FUNCTION_BLOCK Valve
VAR_INPUT
	//configaracionParammetr : configaracionParammetrs;
END_VAR
VAR		
	
	enaNegDir : BOOL := FALSE;
	enaPosDir : BOOL := FALSE;
	command : REAL; // Příkaz -1000 .. 0 .. 1000 [procenta * 10]

	errorDir : BOOL;
	
	currentCommand : REAL := 0;
	prolaz : STRING;
	previousenaNegDir : BOOL; 
	previousenaPosDir : BOOL;
	currentError : BOOL := FALSE; // test error
	
	//command : INT; 
	status : REFERENCE TO Staus REF=generalVariable.staus;
	konfiguraParametry : REFERENCE TO configaracionParammetrs  REF=generalVariable.conParammetr;
	speedRamp : REAL;
	
END_VAR
VAR_OUTPUT
	OutPosDir : REAL := 0 ;	// Výstup v daném směru [mA]
	OutNegDir : REAL := 0 ;	// Výstup v daném směru [mA]
END_VAR

//currentDir := currentDirB(enaNegDir,enaPosDir);
signalStandstill();
prolaz := 'fb';
IF (currentcommand <> command) THEN
		//nTime := elapsTime(direction := currentDir);
		prolaz := 'različiti';
		currentcommand := rampValve ();
	ELSE	
		Accel_Decel(FALSE, FALSE);
		status.bDone := TRUE;
END_IF;

METHOD PRIVATE Accel_Decel
VAR_INPUT
	a : BOOL;
	b : BOOL;
END_VAR
status.Accel := a;
status.Decel := b;
END_METHOD

METHOD addCommand
VAR_INPUT
	comm : real;
END_VAR
command := comm;	
currentError := FALSE;
errorDir := FALSE;
END_METHOD

METHOD PUBLIC commandCheck
VAR_INPUT
	comm : REAL;
END_VAR
VAR
	
END_VAR
IF not(currentError) THEN
	IF ((comm <= 100) AND (comm >0)) THEN
			IF enaPosDir THEN
				addCommand(comm);
			ELSIF NOT(errorDir) THEN
					errCode(4);
					errorDir := TRUE;
				END_IF
		ELSIF ((comm >= -100) AND (comm < 0)) THEN
				IF enaNegDir THEN
					addCommand(comm);
				ELSIF not(errorDir) THEN
					errCode(3);
					errorDir := TRUE;
				END_IF
				ELSIF comm = 0 THEN
						status.Standstill := 0;
						addCommand(comm);
					ELSIF NOT(errorDir) THEN
					errCode(2);
					errorDir := TRUE;
				END_IF
END_IF
END_METHOD

METHOD PRIVATE convertTo : REAL
VAR_INPUT
	currCommand : REAL;
END_VAR
IF enaPosDir THEN
	convertTo := 100*(currCommand -konfiguraParametry.CurPosDirMin)/(konfiguraParametry.CurPosDirMax - konfiguraParametry.CurPosDirMin);
ELSE
	convertTo := 100*(currCommand -konfiguraParametry.CurNegDirMin)/(konfiguraParametry.CurnegDirMax - konfiguraParametry.CurNegDirMin);
END_IF
END_METHOD

METHOD PROTECTED convertToAnal : REAL
VAR_INPUT
	pCommand : REAL;
END_VAR
IF  enaPosDir THEN
	convertToAnal:= (pCommand * (konfiguraParametry.CurPosDirMax - konfiguraParametry.CurPosDirMin)/1000) + konfiguraParametry.CurPosDirMin;
ELSE
	convertToAnal:= (pCommand * (konfiguraParametry.CurNegDirMax - konfiguraParametry.CurNegDirMin)/1000) + konfiguraParametry.CurNegDirMin;
END_IF
END_METHOD

METHOD PRIVATE elapsTime : REAL
VAR_INPUT
	direction : BOOL;
END_VAR
IF direction THEN
		elapsTime := (konfiguraParametry.CurPosDirMax - konfiguraParametry.CurPosDirMin)/(konfiguraParametry.RampPosDirDown -konfiguraParametry.RampPosDirUp);
	ELSE
		elapsTime := (konfiguraParametry.CurNegDirMax - konfiguraParametry.CurNegDirMin)/(konfiguraParametry.RampNegDirDown -konfiguraParametry.RampNegDirUp);
END_IF
END_METHOD

METHOD PUBLIC enableSolenoidControl
VAR_INPUT
	poz : BOOL;
	neg : BOOL;	
END_VAR
IF (poz AND neg) THEN
	// error 
	errCode(1);
	ELSE
	enaNegDir := neg;
	enaPosDir := poz;
	currentError := FALSE ;
END_IF
END_METHOD

METHOD PRIVATE errCode
VAR_INPUT
	ErrorId : INT; // Kód chyby
END_VAR

CASE ErrorId OF
		1: messageError('muze byt aktivní pouze jedna cívka (PosDir nebo NegDir)');
		2: messageError('hodnot od -100 .. 0 .. 100');
		3: messageError('enable Negativ is False');
		4: messageError('enable Poszitive is False');
		5: messageError('nemuže enable Pos a Neg spolu');
	END_CASE
status.nErrorId := ErrorId;
END_METHOD

METHOD PRIVATE messageError 
VAR_INPUT
	sError :STRING;
END_VAR
IF NOT(currentError) THEN
	status.bError := sError;
	blockMessage(error := sError);
	currentError := TRUE;
END_IF
END_METHOD

METHOD PRIVATE rampTimeCalculate : REAL
VAR_INPUT
	cMax : REAL;
	cMin : REAL;
	rampDirTime : INT;
	delta : real;
END_VAR
rampTimeCalculate := abs(delta / (cMax -cMin)/ rampDirTime);
END_METHOD

METHOD PRIVATE rampTimeDown : INT
VAR_INPUT
END_VAR
//RampTimePosDirUp = (configaracionParammetr.CurPosDirMax - configaracionParammetr.CurPosDirMin) / (configaracionParammetr.RampPosDirUp - Deadtime);
END_METHOD

METHOD PRIVATE rampValve : REAL
VAR_INPUT
END_VAR
VAR
	mAcurrentCommand : REAL; 
	mAcommand : REAL;
	delta : REAL;
	rateTime : REAL;
	direction : INT;
END_VAR
prolaz := 'UPAO u rampvalme';
status.Standstill := FALSE;	
IF enaNegDir THEN
	prolaz := 'negTIVNI';
	direction := -1;
	ELSIF enaPosDir THEN
		prolaz := 'pozitivni';
		direction := 1;
END_IF
delta :=  ABS(command) - ABS(currentCommand);
mAcurrentCommand := direction * convertToAnal(currentCommand*10);
mAcommand := direction * convertToAnal(command*10);

IF (currentCommand * command) >= 0 THEN
		// iste znak 
		prolaz := 'isti znak';
					
		IF (delta > 0 ) THEN
			// raste
			prolaz := 'delata veći od 0 ';
			//pitanje da li je dozvola uključena
			
			IF (enaNegDir XOR enaPosDir) THEN
				Accel_Decel(TRUE , FALSE);
				prolaz := 'raste';
				IF (enaPosDir AND command > 0) THEN
						rateTime := rampValveDirection(delta, 1);
					ELSIF (enaNegDir AND command <0) THEN
							rateTime := rampValveDirection(delta, 2);
						ELSE
							command := 0;
				END_IF;
			END_IF;
				mAcurrentCommand := accelerationValve(mAcurrentCommand, mAcommand, rateTime);
		ELSE
			// opada
			prolaz := 'opada';
			Accel_Decel(FALSE , TRUE);
			IF enaNegDir THEN
				rateTime := rampValveDirection(delta, 3);
				ELSE
				rateTime := rampValveDirection(delta, 4);
			END_IF;
			mAcurrentCommand := decelerationValve(mAcurrentCommand, mAcommand, rateTime);
		END_IF;
ELSE
		// različiti znakovi	->	prvo opada
		IF enaNegDir THEN
			rateTime := rampValveDirection(delta, 3);
		ELSE
			rateTime := rampValveDirection(delta, 4);
		END_IF;
		Accel_Decel(FALSE , TRUE);
		mAcurrentCommand := decelerationValve(mAcurrentCommand, 0, rateTime);
END_IF;
	 
	IF (mAcurrentCommand = 0) THEN
		OutNegDir := 0;
		OutPosDir := 0;
		waitbDeathtime();
		ELSIF enaPosDir > 0 THEN
			OutPosDir := mAcurrentCommand;
			OutNegDir := 0;
			ELSE
				OutNegDir := mAcurrentCommand;
				OutPosDir := 0;
		END_IF;
			
rampValve := direction * convertTo(mAcurrentCommand);
END_METHOD

METHOD PRIVATE rampValveDirection : REAL
VAR_INPUT
	delta : REAL;
	i :INT;
END_VAR
CASE i OF
	1:	//Pos  addd
		rampValveDirection := rampTimeCalculate(konfiguraParametry.CurPosDirMax, konfiguraParametry.CurPosDirMin, konfiguraParametry.RampNegDirUp ,delta);
	2: 	//Neg add
		rampValveDirection := rampTimeCalculate(konfiguraParametry.CurNegDirMax, konfiguraParametry.CurNegDirMin, konfiguraParametry.RampNegDirUp ,delta);
	3: 	//pos dec
		rampValveDirection := rampTimeCalculate(konfiguraParametry.CurPosDirMin, konfiguraParametry.CurPosDirMax, konfiguraParametry.RampNegDirDown ,delta);
	4: 	//neg dec
		rampValveDirection := rampTimeCalculate(konfiguraParametry.CurNegDirMin, konfiguraParametry.CurNegDirMax, konfiguraParametry.RampNegDirDown ,delta);
END_CASE
END_METHOD

METHOD signalbBussy : BOOL
VAR_INPUT
END_VAR
END_METHOD

METHOD signalOutDirProc 
VAR_INPUT
	signalOutDirProc : REAL;
END_VAR
VAR_OUTPUT
	OutNegDirProc : REAL;
	OutPosDirProc : real;
END_VAR
signalOutDirProc := command;
IF (signalOutDirProc > 0) THEN
	OutNegDirProc := signalOutDirProc;
	ELSE
		OutPosDirProc := signalOutDirProc;
	END_IF
END_METHOD

METHOD PRIVATE signalStandstill : BOOL
IF (OutPosDir = OutNegDir = 0) THEN
	status.Standstill := TRUE;
	ELSE
		status.Standstill := FALSE;
END_IF
END_METHOD

METHOD PRIVATE speedRampValve 
VAR_INPUT
	i: INT;
END_VAR
// speed Valve transition  Max to min and reverse
CASE i OF
	1 : speedRamp := (konfiguraParametry.CurNegDirMin)/konfiguraParametry.RampNegDirUp;
	2 : speedRamp := (konfiguraParametry.CurNegDirMin)/konfiguraParametry.RampNegDirDown;
	3 : speedRamp := (konfiguraParametry.CurPosDirMin)/konfiguraParametry.RampPosDirUp;
	4 : speedRamp := (konfiguraParametry.CurPosDirMin)/konfiguraParametry.RampPosDirDown;
END_CASE
END_METHOD

METHOD Standstill 
VAR_INPUT
END_VAR
IF (command = 0 ) THEN
	status.Standstill := TRUE;
	blockMessage('Oba výstupy jsou na minimum');
END_IF
END_METHOD

METHOD waitbDeathtime : BOOL
VAR
	delay : TON;
	dTime : TIME;
END_VAR
dTime := INT_TO_TIME(generalVariable.conParammetr.Deadtime);
delay(IN := TRUE, PT:= dtime);
            IF NOT (delay.Q) THEN
                RETURN;
            END_IF;

delay(IN := FALSE);
END_METHOD

END_FUNCTION_BLOCK

(* stored: Version 1.1.0.1, ProductVersion 3.1.4024.12
   POU Valve: Id {07fe6f2a-6d45-441b-87af-c7e504d72a69}, SpecialFunc None
   Folder convert: Id {300b4007-52ce-45a9-b54b-66603ed0f738}
   Folder status: Id {c3096d7a-3e5f-4ec9-98f8-fe780d20a6f1}
   Method Accel_Decel: Id {5fabbdb6-e851-4631-9979-90e5066b5d5d}
   Method addCommand: Id {6c3d938e-09ec-4b69-ab31-3c4b3a35ae7e}
   Method commandCheck: Id {ea8fb27c-a143-4ddf-a1d6-d37603ca1158}
   Method convertTo: Id {71dc1983-f851-4477-9ad3-772e0d3c40e3}
   Method convertToAnal: Id {ef17a997-e61a-4973-93d5-edbe7345e470}
   Method elapsTime: Id {942fb0ec-ddb1-47fe-a405-090f8689464c}
   Method enableSolenoidControl: Id {bc641138-3214-4040-8ffb-ac7a51b96b0e}
   Method errCode: Id {5db0075d-b956-4fda-a9b7-ef361dbb8a72}
   Method messageError: Id {30631b2c-d480-418c-b15e-5ad6737037e0}
   Method rampTimeCalculate: Id {141d03d7-0681-44d0-8863-fc4051283fe9}
   Method rampTimeDown: Id {64b1fda7-6a13-4ee0-a012-61c688c72f68}
   Method rampValve: Id {efb1c5bc-55a9-4dd2-9df6-4eaae4ba8546}
   Method rampValveDirection: Id {52938cef-64ef-46fe-9bb3-0b93254c1a51}
   Method signalbBussy: Id {24c66bc9-cbea-473d-a7b9-0ec9e7977592}
   Method signalOutDirProc: Id {cbe8e172-7050-478d-b9ce-04bc75d3051f}
   Method signalStandstill: Id {85d95741-4973-493f-b221-ce79aefa42c8}
   Method speedRampValve: Id {715f72a7-690c-4176-8487-a38148e045c1}
   Method Standstill: Id {0645a22c-46c8-4c4c-93ad-b7dded02cf14}
   Method waitbDeathtime: Id {b79e3e4c-d012-4eb0-bcad-6964bfc150a0} *)
